Fanuc TP program (LS listing): ros.ls

/PROG  ROS
/ATTR
OWNER		= MNEDITOR;
COMMENT		= "r4:krl_moveto";
PROG_SIZE	= 152;
CREATE		= DATE 12-10-02  TIME 12:09:14;
MODIFIED	= DATE 12-10-02  TIME 12:09:14;
FILE_NAME	= ;
VERSION		= 0;
LINE_COUNT	= 2;
MEMORY_SIZE	= 500;
PROTECT		= READ_WRITE;
TCD:  STACK_SIZE	= 0,
      TASK_PRIORITY	= 50,
      TIME_SLICE	= 0,
      BUSY_LAMP_OFF	= 0,
      ABORT_REQUEST	= 0,
      PAUSE_REQUEST	= 7;
DEFAULT_GROUP	= *,*,*,*,*;
CONTROL_CODE	= 00000000 00000000;
/MN
   1:  CALL TASK_RUN('ROS_S') ;
   2:  CALL ROS_R    ;
/POS
/END
